FUNCTION_BLOCK AB_CMDPARSER (* Basic FB with empty ECC *)
  (* Standard: 61499-2 *)
  (* Version 1.0, 2023-01-19, Alex Maximov *)
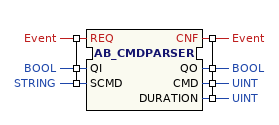
  EVENT_INPUT
    REQ WITH QI, SCMD;
  END_EVENT
  EVENT_OUTPUT
    CNF WITH QO, CMD, DURATION;
  END_EVENT
  VAR_INPUT
    QI : BOOL;
    SCMD : STRING;
  END_VAR
  VAR_OUTPUT
    QO : BOOL;
    CMD : UINT;
    DURATION : UINT;
  END_VAR
  EC_STATES
    START; (* Initial State *)
  END_STATES
END_FUNCTION_BLOCK
